KUKA KRL data list: STRING_FROM_BUS.dat

&ACCESS RV
&PARAM TEMPLATE = C:\KRC\Roboter\Template\vorgabe
&PARAM EDITMASK = *
DEFDAT string_from_bus

GLOBAL CHAR gsStringFromBus[60] = " "

ENDDAT
